// Mitsubishi GX Works2 project: PLC_GROUP_10   PLC: FX3G

// global labels: Global1
VAR_GLOBAL CONSTANT
  spieces_ratio : REAL := 0.1;
END_VAR
VAR_GLOBAL
  spieces_wanted AT D1118 : REAL;
  oil_wanted AT D1114 : REAL;
  water_wanted AT D1116 : REAL;
  yeast_wanted AT D1112 : REAL;
  Enough_yeast AT M11 : BOOL;
  Enough_oil AT M12 : BOOL;
  Enough_spieces AT M14 : BOOL;
  turn_of_flickering AT TC1 : BOOL;
END_VAR
VAR_GLOBAL CONSTANT
  ThreeSec : INT := 30;
END_VAR
VAR_GLOBAL
  blink AT M5 : BOOL;
  TC2 AT TC2 : BOOL;
  TC_2 AT TC2 : BOOL;
END_VAR
VAR_GLOBAL CONSTANT
  half_Sec : INT := 5;
END_VAR
VAR_GLOBAL
  TS_2 AT TS2 : BOOL;
  TC_3 AT TC3 : BOOL;
  TS_3 AT TS3 : BOOL;
  TS_1 AT TS1 : BOOL;
  StatrWork AT X002 : BOOL;
  StartWork AT X002 : BOOL;
  TS_5 AT TS5 : BOOL;
END_VAR
VAR_GLOBAL CONSTANT
  Lamp_on : REAL := 30.0;
END_VAR
VAR_GLOBAL
  TC_5 AT TC5 : BOOL;
  Lamp_Before_work AT Y005 : BOOL;
END_VAR
VAR_GLOBAL CONSTANT
  const100 : REAL := 100.0;
END_VAR
VAR_GLOBAL
  Kneading_flour AT D1300 : REAL;
END_VAR
VAR_GLOBAL CONSTANT
  const20 : REAL := 20.0;
END_VAR
VAR_GLOBAL
  Kneading_yeast AT D1302 : REAL;
END_VAR
VAR_GLOBAL CONSTANT
  const50 : REAL := 50.0;
END_VAR
VAR_GLOBAL
  Kneading_water AT D1306 : REAL;
END_VAR
VAR_GLOBAL CONSTANT
  const30 : REAL := 30.0;
END_VAR
VAR_GLOBAL
  Kneading_oil AT D1304 : REAL;
  Kneading_spieces AT D1308 : REAL;
END_VAR
VAR_GLOBAL CONSTANT
  const10 : REAL := 10.0;
END_VAR
VAR_GLOBAL
  TC_4 AT TC4 : BOOL;
  TS_4 AT TS4 : BOOL;
  Start_kneading AT X001 : BOOL;
  kneading_light AT Y001 : BOOL;
  mix_flour AT D1300 : REAL;
  mix_yeast AT D1302 : REAL;
  mix_water AT D1306 : REAL;
  mix_oil AT D1304 : REAL;
  mix_spieces AT D1308 : REAL;
  rising_flour AT D1400 : REAL;
  rising_yeast AT D1402 : REAL;
  rising_water AT D1406 : REAL;
  rising_oil AT D1404 : REAL;
  rising_spieces AT D1408 : REAL;
  Start_baking AT M9 : BOOL;
  Start_rising AT M100 : BOOL;
  baking_flour AT D1500 : REAL;
  baking_yeast AT D1502 : REAL;
  baking_water AT D1506 : REAL;
  baking_oil AT D1504 : REAL;
  baking_spieces AT D1508 : REAL;
  Start_Mix AT X001 : BOOL;
  Mix_light AT Y001 : BOOL;
  Start_Rising_Dough AT X011 : BOOL;
  Count_Clicks AT CC1 : BOOL;
END_VAR
VAR_GLOBAL CONSTANT
  clicks_2 : INT := 2;
END_VAR
VAR_GLOBAL
  CS_1 AT CS1 : BOOL;
  turn_of_blinking AT TC8 : BOOL;
  TC_8 AT TC8 : BOOL;
  blinking AT M7 : BOOL;
  TC_6 AT TC6 : BOOL;
  TS_6 AT TS6 : BOOL;
  Rising_Light_1 AT Y002 : BOOL;
  TC_7 AT TC7 : BOOL;
  TS_7 AT TS7 : BOOL;
  Rising_Light_2 AT Y003 : BOOL;
  TS_8 AT TS8 : BOOL;
  finish_Raising AT M8 : BOOL;
  finish_Rising AT M8 : BOOL;
  TS_9 AT TS9 : BOOL;
  baking AT Y004 : BOOL;
  EnoughStock AT M2 : BOOL;
  Transfer_ingridients AT M13 : BOOL;
  flour_trasfered AT M15 : BOOL;
  yeast_trasfered AT M16 : BOOL;
  water_trasfered AT M17 : BOOL;
  oil_trasfered AT M18 : BOOL;
  spieces_trasfered AT M19 : BOOL;
  Start_clock AT M20 : BOOL;
  TransferFlour AT M21 : BOOL;
  TransferYeast AT M22 : BOOL;
  TrasnferWater AT M22 : BOOL;
  TransferOil AT M24 : BOOL;
  TransferWater AT M23 : BOOL;
  TransferSpeices AT M25 : BOOL;
  TransferIngridients AT M80 : BOOL;
  StartClock AT M26 : BOOL;
  baking_timer AT TC9 : BOOL;
  TrayonShelf_flour AT D1600 : REAL;
  TrayonShelf_yeast AT D1602 : REAL;
  TrayonShelf_water AT D1606 : REAL;
  TrayonShelf_oil AT D1604 : REAL;
  TrayonShelf_spieces AT D1608 : REAL;
  Transfer_Flour AT M26 : BOOL;
  Transfer_Yeast AT M27 : BOOL;
  Transfer_Water AT M28 : BOOL;
  Transfer_Oil AT M29 : BOOL;
  Transfer_Speices AT M30 : BOOL;
  quality_check AT X003 : BOOL;
  Check_amounts AT CC16 : BOOL;
END_VAR
VAR_GLOBAL CONSTANT
  two_checks : INT := 3;
END_VAR
VAR_GLOBAL
  CS_2 AT CS2 : BOOL;
  Analog_Input_2 AT D8281 : REAL;
END_VAR
VAR_GLOBAL CONSTANT
  LB : INT := 400;
END_VAR
VAR_GLOBAL
  GE_than_1 AT M27 : BOOL;
  LE_than_5 AT M28 : BOOL;
  quality_timer AT TC11 : BOOL;
END_VAR
VAR_GLOBAL CONSTANT
  five_sec : INT := 50;
  UB : INT := 2000;
END_VAR
VAR_GLOBAL
  TS_11 AT TS11 : BOOL;
  quality_light AT Y006 : BOOL;
  ThrowToGarbage AT M30 : BOOL;
END_VAR
VAR_GLOBAL CONSTANT
  const0 : REAL;
  oil_ratio : REAL := 0.3;
  water_ratio : REAL := 0.5;
  yeast_ratio : REAL := 0.2;
  constant_100 : REAL := 100.0;
END_VAR
VAR_GLOBAL
  OutOfStock AT M2 : BOOL;
  EmergencyButton AT X007 : BOOL;
  EndWorkDay AT M10 : BOOL;
  WorkDayLight AT Y010 : BOOL;
  StartDay AT X010 : BOOL;
  spices_stock AT D1208 : REAL;
  spieces_input AT D1108 : REAL;
  spieces_stock AT D1208 : REAL;
  sesame_stock AT D1212 : REAL;
  sesame_input AT D1114 : REAL;
  salt_stock AT D1210 : REAL;
  salt_input AT D1112 : REAL;
  suger_stock AT D1208 : REAL;
  suger_input AT D1110 : REAL;
  water_stock AT D1206 : REAL;
  water_input AT D1106 : REAL;
  oil_stock AT D1204 : REAL;
  oil_input AT D1104 : REAL;
  yeast_stock AT D1202 : REAL;
  yeast_input AT D1102 : REAL;
  flour_input AT D1100 : REAL;
  flour_stock AT D1200 : REAL;
  Switch_start_Day AT X010 : BOOL;
  Lamp_start_work AT Y005 : BOOL;
  Switch1 AT X002 : BOOL;
  Enough_water AT M13 : BOOL;
END_VAR
VAR_GLOBAL CONSTANT
  four_sec : INT := 40;
END_VAR
VAR_GLOBAL
  Steady_light AT M50 : BOOL;
  blinking_light AT M51 : BOOL;
  Mix_active AT M60 : BOOL;
  Counter_light AT M61 : BOOL;
  off_blinkingLight AT M52 : BOOL;
  Check1 AT M80 : BOOL;
  Check2 AT M81 : BOOL;
  Check3 AT M82 : BOOL;
  Check4 AT M83 : BOOL;
  Check5 AT M84 : BOOL;
  yalla AT M100 : BOOL;
  SHAY AT M222 : BOOL;
  closed AT M223 : BOOL;
  RESET_DAY AT M224 : BOOL;
  AnalogInput2 AT D8281 : INT;
END_VAR
VAR_GLOBAL CONSTANT
  LBLB : REAL := 2000.0;
END_VAR
VAR_GLOBAL
  ResetCounter AT M230 : BOOL;
  REalinput AT D8281 : REAL;
  CC_2 AT CC2 : BOOL;
  LB_flour AT M102 : BOOL;
END_VAR
VAR_GLOBAL CONSTANT
  two_checks_forGarbage : INT := 2;
END_VAR
VAR_GLOBAL
  CC_3 AT CC3 : BOOL;
  M_Flour AT M338 : BOOL;
  M_Yeast AT M339 : BOOL;
  M_Water AT M340 : BOOL;
  M_Oil AT M341 : BOOL;
  M_Spieces AT M342 : BOOL;
  M_Flour2 AT M330 : BOOL;
  M_Yeast2 AT M331 : BOOL;
  M_Wate2r AT M332 : BOOL;
  M_Oil2 AT M333 : BOOL;
  M_Spieces2 AT M334 : BOOL;
  M_Wate2 AT M332 : BOOL;
  M_Water2 AT M332 : BOOL;
  finish_it AT M335 : BOOL;
  flour_container AT D1250 : REAL;
  yeast_container AT D1252 : REAL;
  water_container AT D1256 : REAL;
  oil_container AT D1254 : REAL;
  spieces_container AT D1258 : REAL;
  Lamp_Y5Off AT M288 : BOOL;
  UB_twoChecks AT CC2 : BOOL;
  twoChecksForGarbage AT CC3 : BOOL;
  quality_const AT M20 : BOOL;
END_VAR

// task Task_01 (event TRUE, interval 0, priority 31): POU_01

PROGRAM POU_01
(* structured ladder/FBD written out as ST: instructions are called as NAME(EN, inputs, outputs); _pN, _eN, _tN stand for wires *)
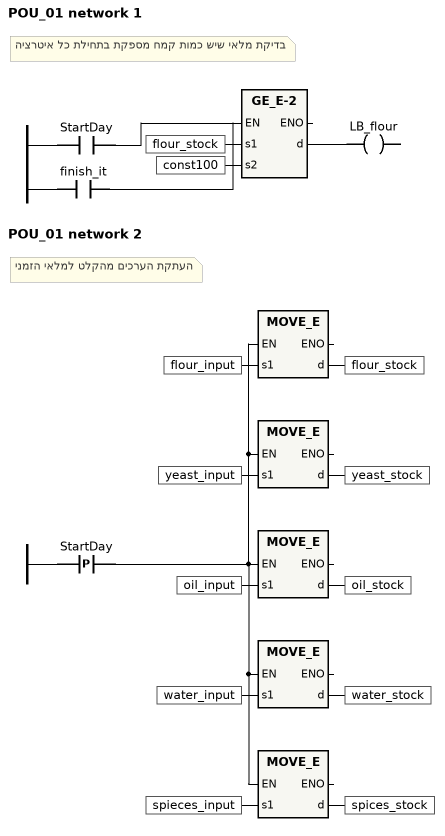
(* network 1 *)
(* בדיקת מלאי שיש כמות קמח מספקת בתחילת כל איטרציה *)
GE_E(StartDay OR finish_it, flour_stock, const100, _t1);
LB_flour := _t1;
(* network 2 *)
(* העתקת הערכים מהקלט למלאי הזמני *)
_p1 := LDP(TRUE, StartDay);
MOVE_E(_p1, flour_input, flour_stock);
MOVE_E(_p1, yeast_input, yeast_stock);
MOVE_E(_p1, oil_input, oil_stock);
MOVE_E(_p1, water_input, water_stock);
MOVE_E(_p1, spieces_input, spices_stock);
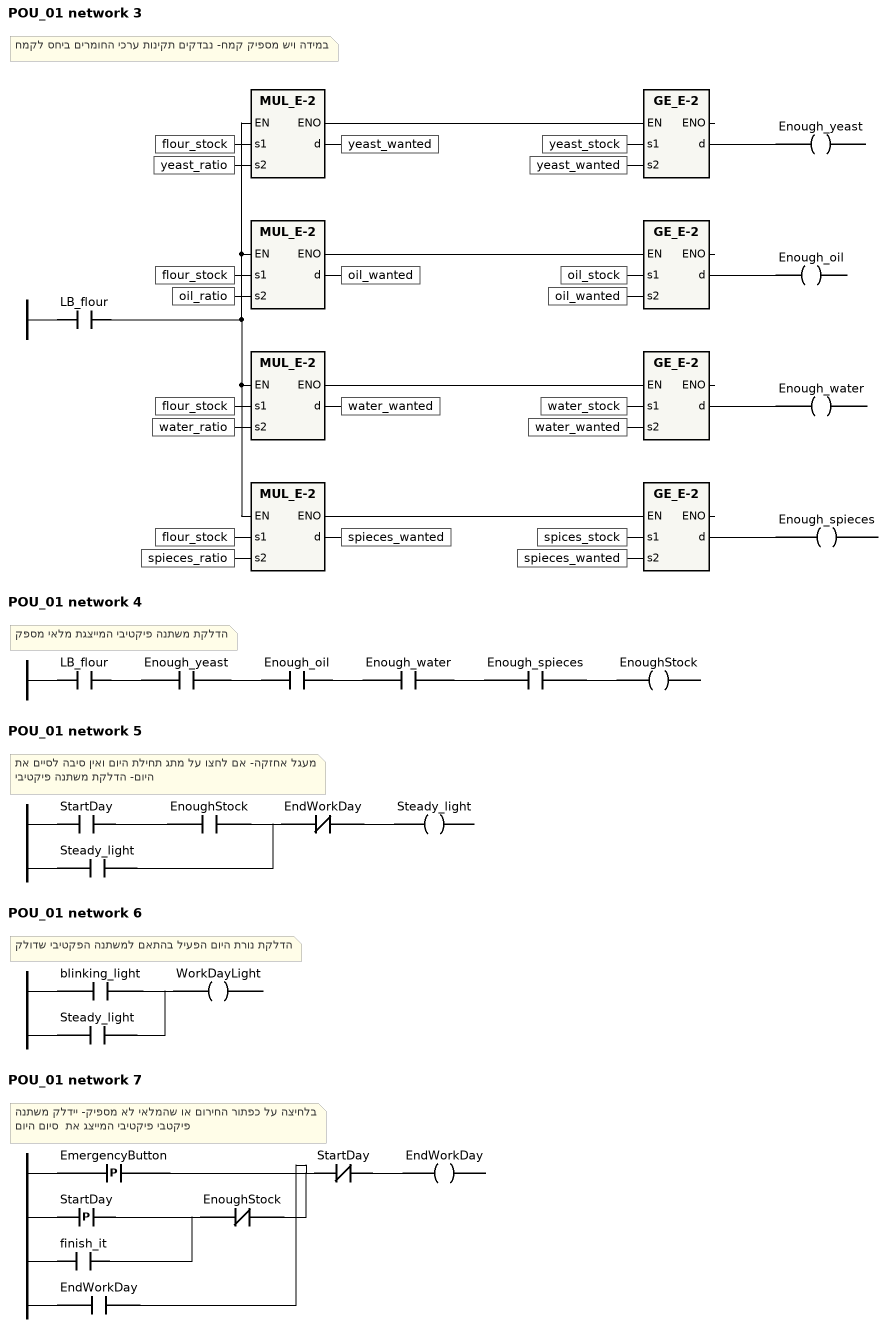
(* network 3 *)
(* במידה ויש מספיק קמח- נבדקים תקינות ערכי החומרים ביחס לקמח *)
_e1 := MUL_E(LB_flour, flour_stock, yeast_ratio, yeast_wanted);
GE_E(_e1, yeast_stock, yeast_wanted, _t2);
Enough_yeast := _t2;
_e3 := MUL_E(LB_flour, flour_stock, oil_ratio, oil_wanted);
GE_E(_e3, oil_stock, oil_wanted, _t4);
Enough_oil := _t4;
_e5 := MUL_E(LB_flour, flour_stock, water_ratio, water_wanted);
GE_E(_e5, water_stock, water_wanted, _t6);
Enough_water := _t6;
_e7 := MUL_E(LB_flour, flour_stock, spieces_ratio, spieces_wanted);
GE_E(_e7, spices_stock, spieces_wanted, _t8);
Enough_spieces := _t8;
(* network 4 *)
(* הדלקת משתנה פיקטיבי המייצגת מלאי מספק *)
EnoughStock := LB_flour AND Enough_yeast AND Enough_oil AND Enough_water AND Enough_spieces;
(* network 5 *)
(* מעגל אחזקה- אם לחצו על מתג תחילת היום ואין סיבה לסיים את היום- הדלקת משתנה פיקטיבי *)
Steady_light := ((StartDay AND EnoughStock) OR Steady_light) AND NOT EndWorkDay;
(* network 6 *)
(* הדלקת נורת היום הפעיל בהתאם למשתנה הפקטיבי שדולק *)
WorkDayLight := blinking_light OR Steady_light;
(* network 7 *)
(* בלחיצה על כפתור החירום או שהמלאי לא מספיק- יידלק משתנה פיקטבי פיקטיבי המייצג את  סיום היום *)
EndWorkDay := (LDP(TRUE, EmergencyButton) OR ((LDP(TRUE, StartDay) OR finish_it) AND NOT EnoughStock) OR EndWorkDay) AND NOT StartDay;
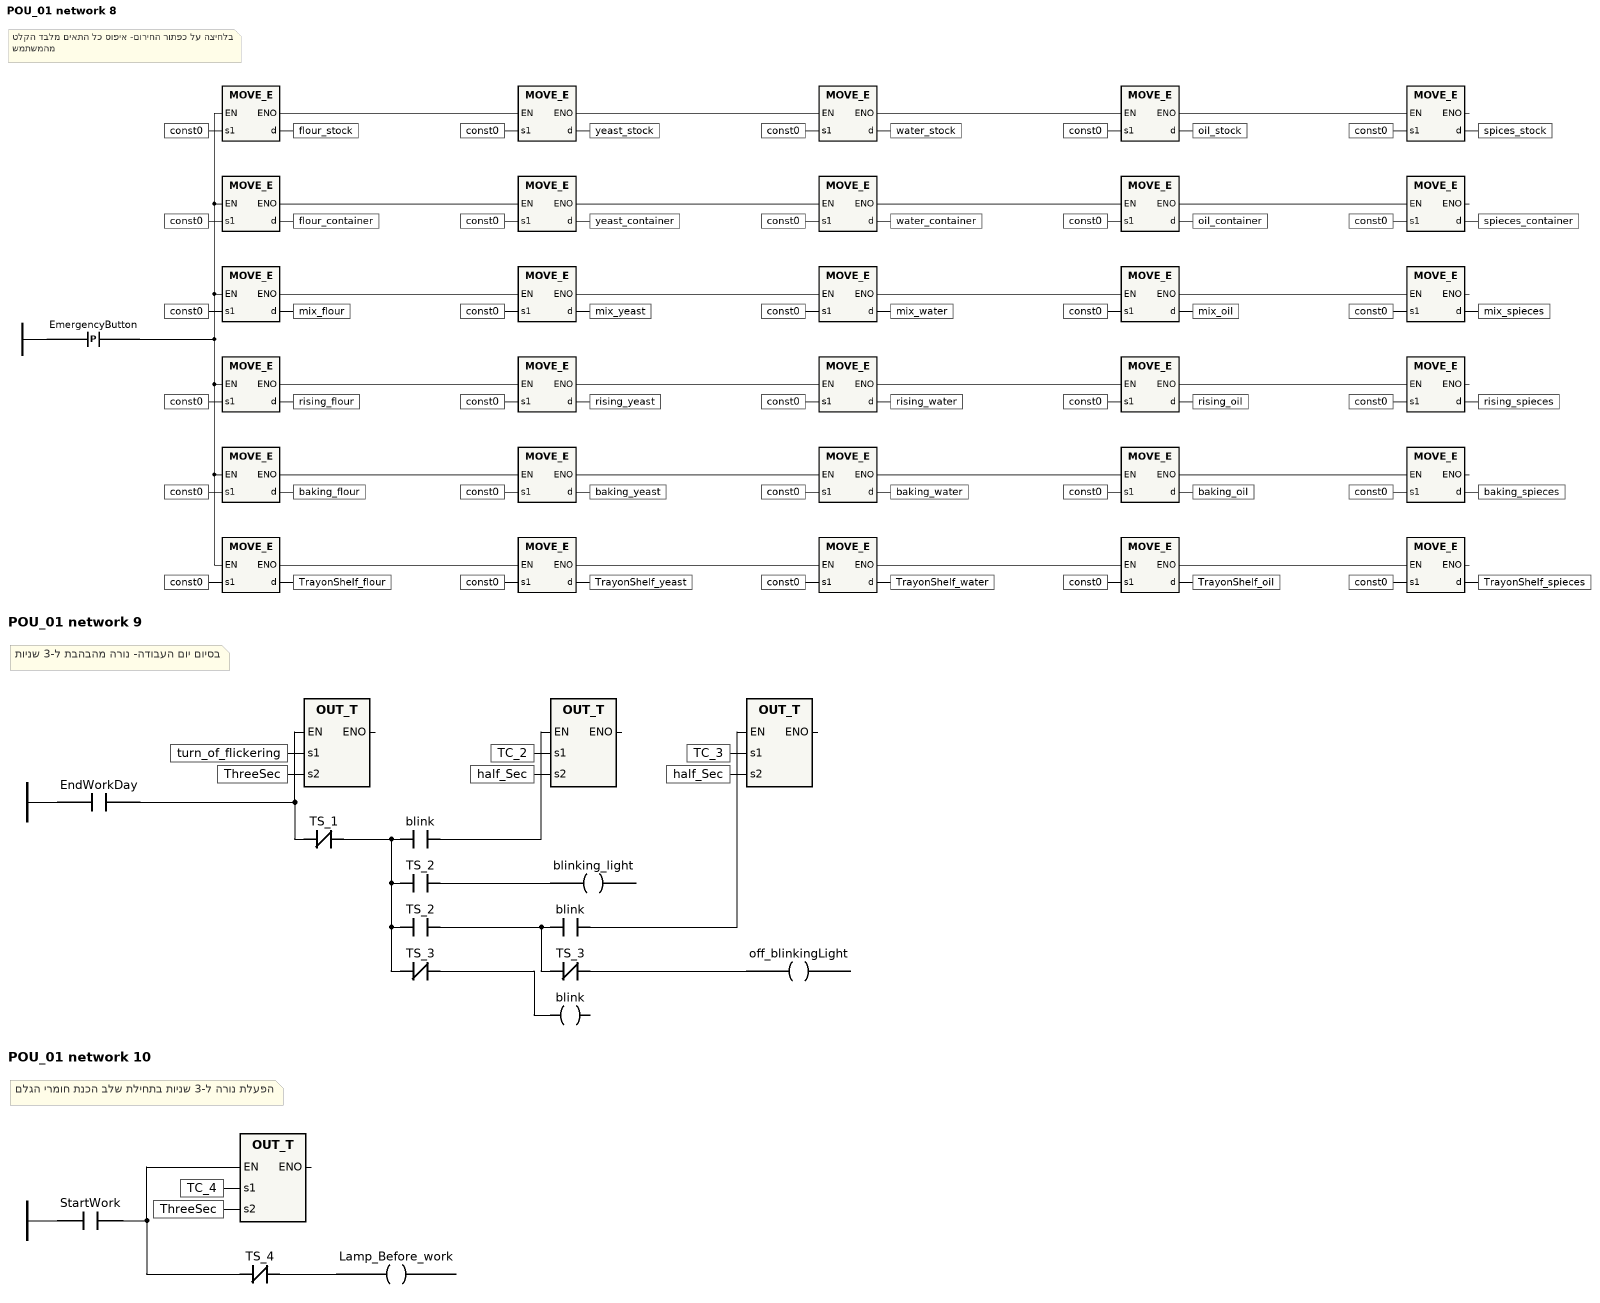
(* network 8 *)
(* בלחיצה על כפתור החירום- איפוס כל התאים מלבד הקלט מהמשתמש *)
_p1 := LDP(TRUE, EmergencyButton);
_e2 := MOVE_E(_p1, const0, flour_stock);
_e3 := MOVE_E(_e2, const0, yeast_stock);
_e4 := MOVE_E(_e3, const0, water_stock);
_e5 := MOVE_E(_e4, const0, oil_stock);
MOVE_E(_e5, const0, spices_stock);
_e6 := MOVE_E(_p1, const0, flour_container);
_e7 := MOVE_E(_e6, const0, yeast_container);
_e8 := MOVE_E(_e7, const0, water_container);
_e9 := MOVE_E(_e8, const0, oil_container);
MOVE_E(_e9, const0, spieces_container);
_e10 := MOVE_E(_p1, const0, mix_flour);
_e11 := MOVE_E(_e10, const0, mix_yeast);
_e12 := MOVE_E(_e11, const0, mix_water);
_e13 := MOVE_E(_e12, const0, mix_oil);
MOVE_E(_e13, const0, mix_spieces);
_e14 := MOVE_E(_p1, const0, rising_flour);
_e15 := MOVE_E(_e14, const0, rising_yeast);
_e16 := MOVE_E(_e15, const0, rising_water);
_e17 := MOVE_E(_e16, const0, rising_oil);
MOVE_E(_e17, const0, rising_spieces);
_e18 := MOVE_E(_p1, const0, baking_flour);
_e19 := MOVE_E(_e18, const0, baking_yeast);
_e20 := MOVE_E(_e19, const0, baking_water);
_e21 := MOVE_E(_e20, const0, baking_oil);
MOVE_E(_e21, const0, baking_spieces);
_e22 := MOVE_E(_p1, const0, TrayonShelf_flour);
_e23 := MOVE_E(_e22, const0, TrayonShelf_yeast);
_e24 := MOVE_E(_e23, const0, TrayonShelf_water);
_e25 := MOVE_E(_e24, const0, TrayonShelf_oil);
MOVE_E(_e25, const0, TrayonShelf_spieces);
(* network 9 *)
(* בסיום יום העבודה- נורה מהבהבת ל-3 שניות *)
OUT_T(EndWorkDay, turn_of_flickering, ThreeSec);
_p1 := EndWorkDay AND NOT TS_1;
OUT_T(_p1 AND blink, TC_2, half_Sec);
blinking_light := _p1 AND TS_2;
_p2 := _p1 AND TS_2;
OUT_T(_p2 AND blink, TC_3, half_Sec);
off_blinkingLight := _p2 AND NOT TS_3;
blink := _p1 AND NOT TS_3;
(* network 10 *)
(* הפעלת נורה ל-3 שניות בתחילת שלב הכנת חומרי הגלם *)
OUT_T(StartWork, TC_4, ThreeSec);
Lamp_Before_work := StartWork AND NOT TS_4;
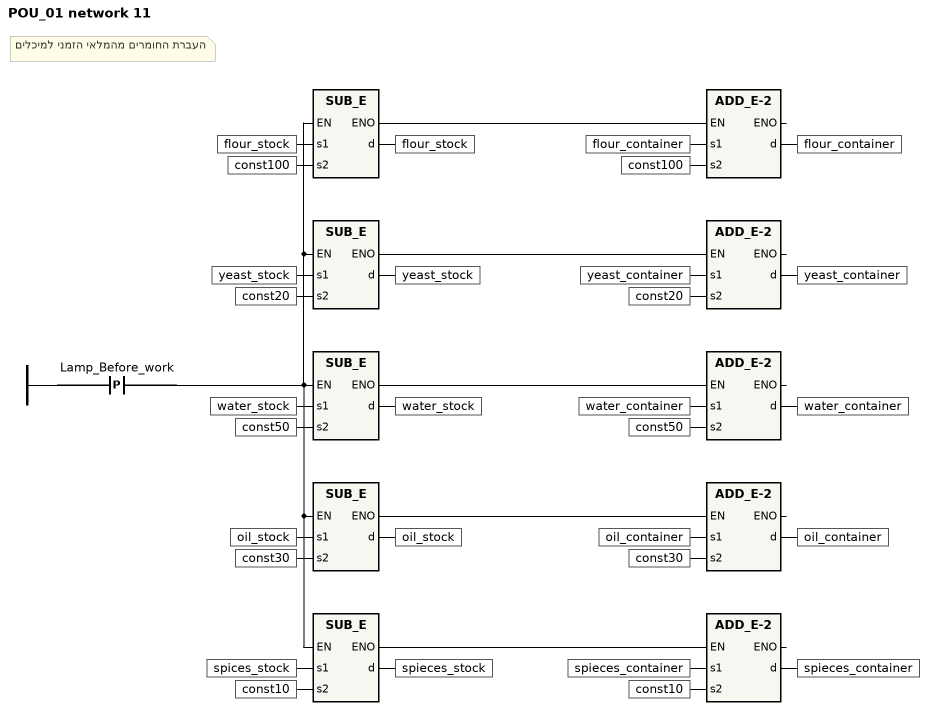
(* network 11 *)
(* העברת החומרים מהמלאי הזמני למיכלים *)
_p1 := LDP(TRUE, Lamp_Before_work);
_e2 := SUB_E(_p1, flour_stock, const100, flour_stock);
ADD_E(_e2, flour_container, const100, flour_container);
_e3 := SUB_E(_p1, yeast_stock, const20, yeast_stock);
ADD_E(_e3, yeast_container, const20, yeast_container);
_e4 := SUB_E(_p1, water_stock, const50, water_stock);
ADD_E(_e4, water_container, const50, water_container);
_e5 := SUB_E(_p1, oil_stock, const30, oil_stock);
ADD_E(_e5, oil_container, const30, oil_container);
_e6 := SUB_E(_p1, spices_stock, const10, spieces_stock);
ADD_E(_e6, spieces_container, const10, spieces_container);
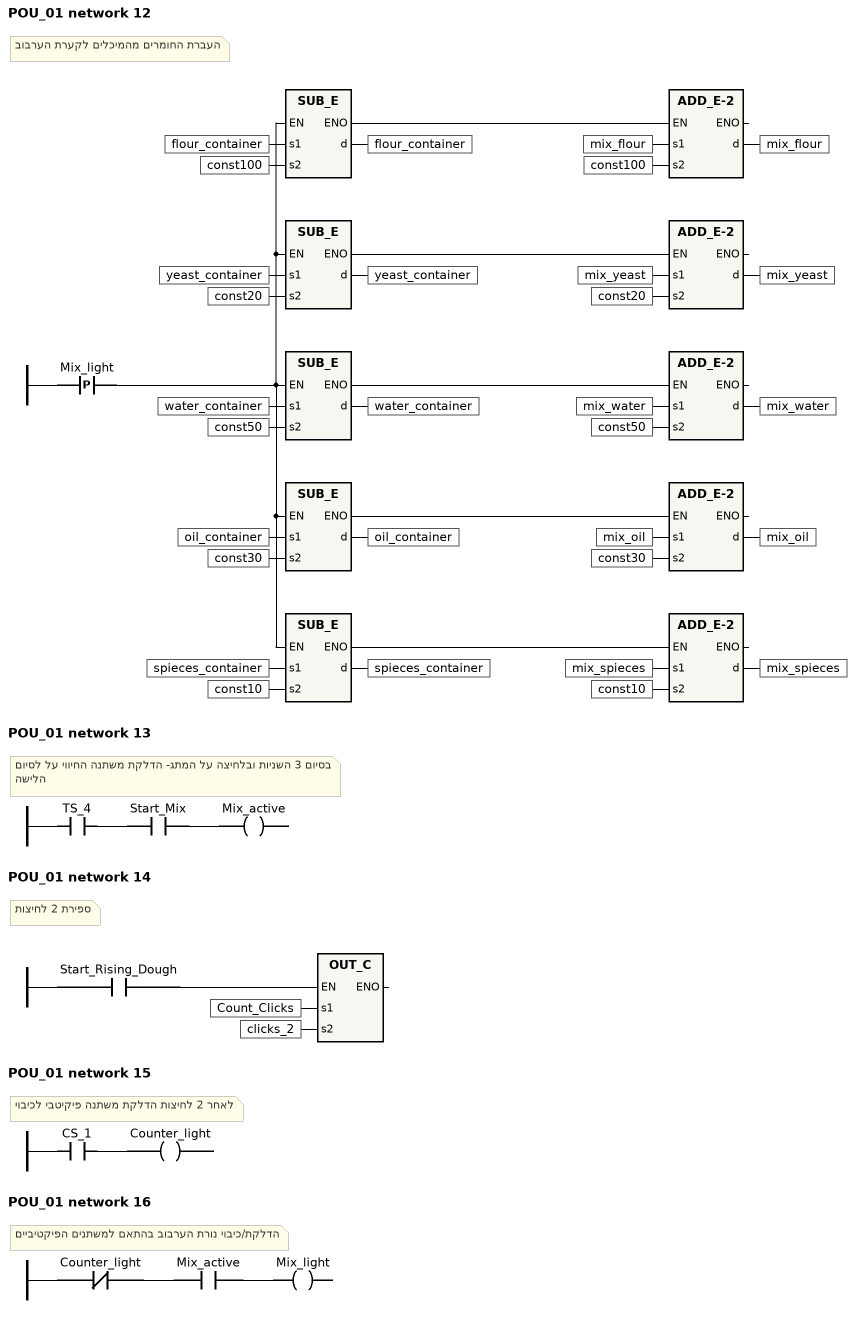
(* network 12 *)
(* העברת החומרים מהמיכלים לקערת הערבוב *)
_p1 := LDP(TRUE, Mix_light);
_e2 := SUB_E(_p1, flour_container, const100, flour_container);
ADD_E(_e2, mix_flour, const100, mix_flour);
_e3 := SUB_E(_p1, yeast_container, const20, yeast_container);
ADD_E(_e3, mix_yeast, const20, mix_yeast);
_e4 := SUB_E(_p1, water_container, const50, water_container);
ADD_E(_e4, mix_water, const50, mix_water);
_e5 := SUB_E(_p1, oil_container, const30, oil_container);
ADD_E(_e5, mix_oil, const30, mix_oil);
_e6 := SUB_E(_p1, spieces_container, const10, spieces_container);
ADD_E(_e6, mix_spieces, const10, mix_spieces);
(* network 13 *)
(* בסיום 3 השניות ובלחיצה על המתג- הדלקת משתנה החיווי על לסיום הלישה *)
Mix_active := TS_4 AND Start_Mix;
(* network 14 *)
(* ספירת 2 לחיצות *)
OUT_C(Start_Rising_Dough, Count_Clicks, clicks_2);
(* network 15 *)
(* לאחר 2 לחיצות הדלקת משתנה פיקיטבי לכיבוי *)
Counter_light := CS_1;
(* network 16 *)
(* הדלקת/כיבוי נורת הערבוב בהתאם למשתנים הפיקטיביים *)
Mix_light := NOT Counter_light AND Mix_active;
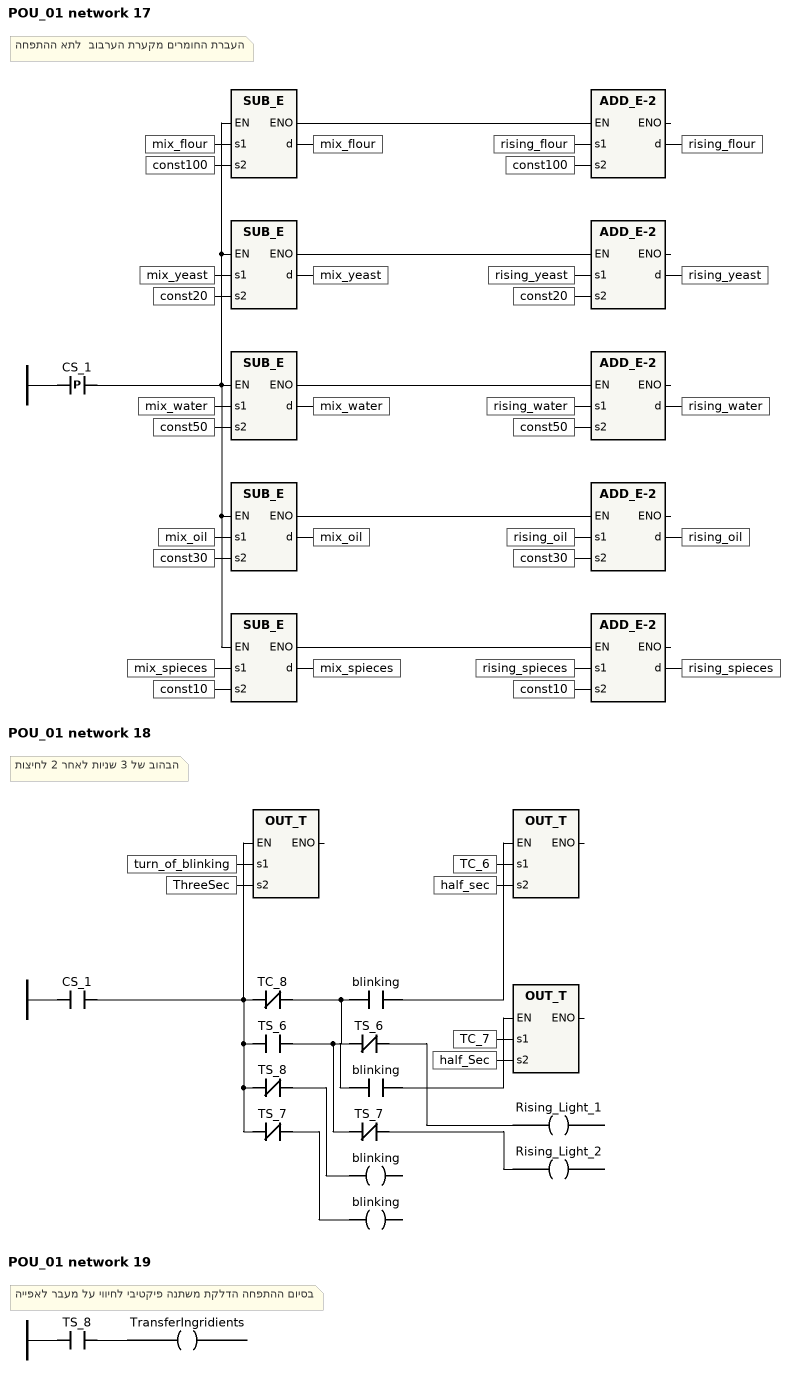
(* network 17 *)
(* העברת החומרים מקערת הערבוב  לתא ההתפחה *)
_p1 := LDP(TRUE, CS_1);
_e2 := SUB_E(_p1, mix_flour, const100, mix_flour);
ADD_E(_e2, rising_flour, const100, rising_flour);
_e3 := SUB_E(_p1, mix_yeast, const20, mix_yeast);
ADD_E(_e3, rising_yeast, const20, rising_yeast);
_e4 := SUB_E(_p1, mix_water, const50, mix_water);
ADD_E(_e4, rising_water, const50, rising_water);
_e5 := SUB_E(_p1, mix_oil, const30, mix_oil);
ADD_E(_e5, rising_oil, const30, rising_oil);
_e6 := SUB_E(_p1, mix_spieces, const10, mix_spieces);
ADD_E(_e6, rising_spieces, const10, rising_spieces);
(* network 18 *)
(* הבהוב של 3 שניות לאחר 2 לחיצות *)
OUT_T(CS_1, turn_of_blinking, ThreeSec);
_p1 := CS_1 AND NOT TC_8;
OUT_T(_p1 AND blinking, TC_6, half_sec);
Rising_Light_1 := _p1 AND NOT TS_6;
_p2 := CS_1 AND TS_6;
OUT_T(_p2 AND blinking, TC_7, half_Sec);
Rising_Light_2 := _p2 AND NOT TS_7;
blinking := CS_1 AND NOT TS_8;
blinking := CS_1 AND NOT TS_7;
(* network 19 *)
(* בסיום ההתפחה הדלקת משתנה פיקטיבי לחיווי על מעבר לאפייה *)
TransferIngridients := TS_8;
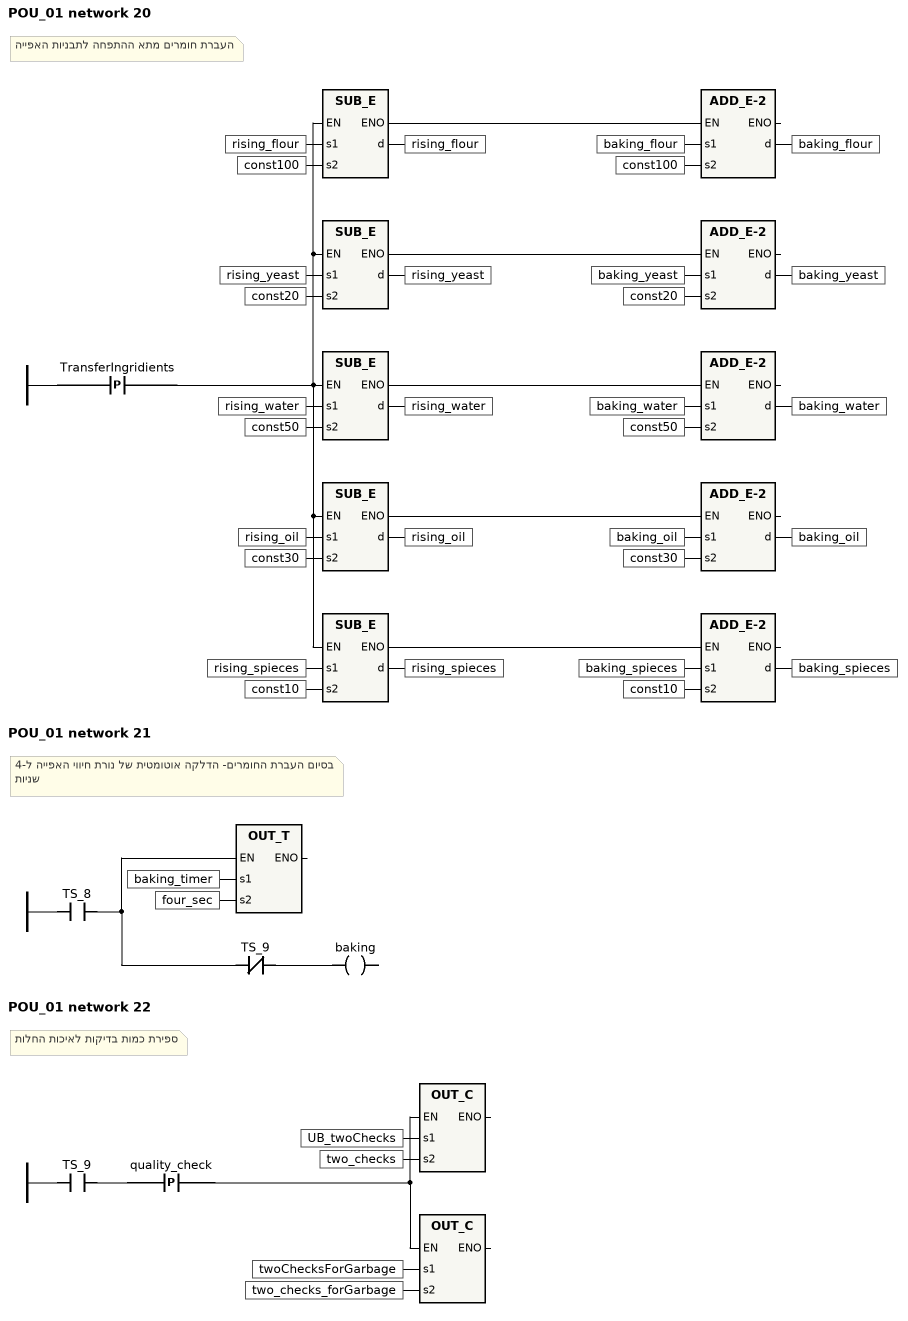
(* network 20 *)
(* העברת חומרים מתא ההתפחה לתבניות האפייה *)
_p1 := LDP(TRUE, TransferIngridients);
_e2 := SUB_E(_p1, rising_flour, const100, rising_flour);
ADD_E(_e2, baking_flour, const100, baking_flour);
_e3 := SUB_E(_p1, rising_yeast, const20, rising_yeast);
ADD_E(_e3, baking_yeast, const20, baking_yeast);
_e4 := SUB_E(_p1, rising_water, const50, rising_water);
ADD_E(_e4, baking_water, const50, baking_water);
_e5 := SUB_E(_p1, rising_oil, const30, rising_oil);
ADD_E(_e5, baking_oil, const30, baking_oil);
_e6 := SUB_E(_p1, rising_spieces, const10, rising_spieces);
ADD_E(_e6, baking_spieces, const10, baking_spieces);
(* network 21 *)
(* בסיום העברת החומרים- הדלקה אוטומטית של נורת חיווי האפייה ל-4 שניות *)
OUT_T(TS_8, baking_timer, four_sec);
baking := TS_8 AND NOT TS_9;
(* network 22 *)
(* ספירת כמות בדיקות לאיכות החלות *)
_p1 := TS_9 AND LDP(TRUE, quality_check);
OUT_C(_p1, UB_twoChecks, two_checks);
OUT_C(_p1, twoChecksForGarbage, two_checks_forGarbage);
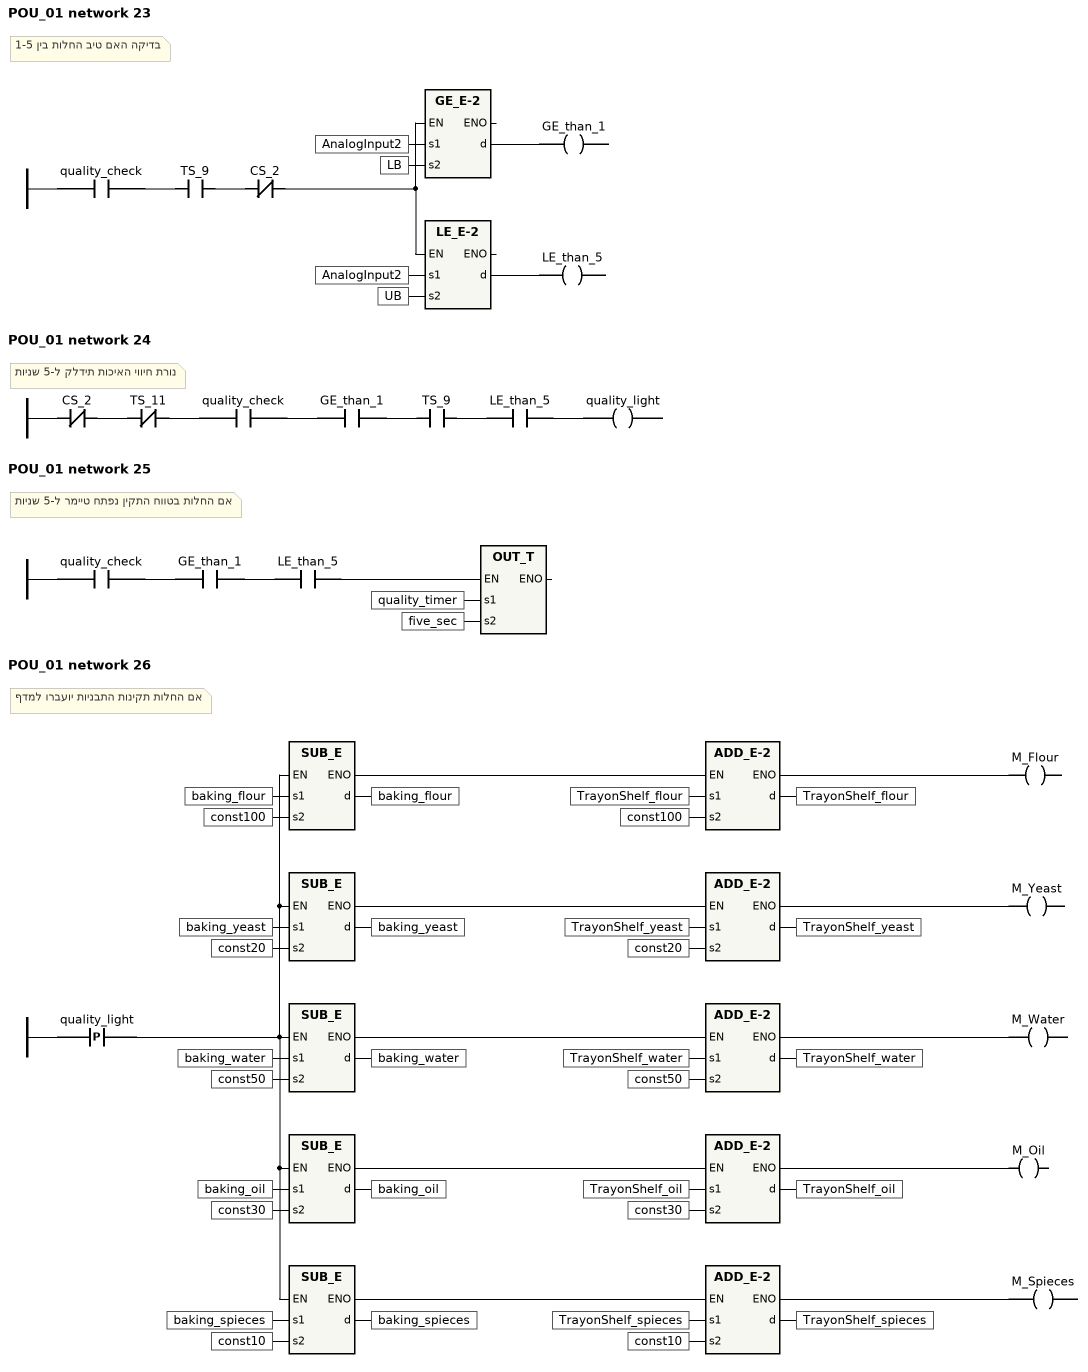
(* network 23 *)
(* בדיקה האם טיב החלות בין 1-5 *)
_p1 := quality_check AND TS_9 AND NOT CS_2;
GE_E(_p1, AnalogInput2, LB, _t2);
GE_than_1 := _t2;
LE_E(_p1, AnalogInput2, UB, _t3);
LE_than_5 := _t3;
(* network 24 *)
(* נורת חיווי האיכות תידלק ל-5 שניות *)
quality_light := NOT CS_2 AND NOT TS_11 AND quality_check AND GE_than_1 AND TS_9 AND LE_than_5;
(* network 25 *)
(* אם החלות בטווח התקין נפתח טיימר ל-5 שניות *)
OUT_T(quality_check AND GE_than_1 AND LE_than_5, quality_timer, five_sec);
(* network 26 *)
(* אם החלות תקינות התבניות יועברו למדף *)
_p1 := LDP(TRUE, quality_light);
_e2 := SUB_E(_p1, baking_flour, const100, baking_flour);
_e3 := ADD_E(_e2, TrayonShelf_flour, const100, TrayonShelf_flour);
M_Flour := _e3;
_e4 := SUB_E(_p1, baking_yeast, const20, baking_yeast);
_e5 := ADD_E(_e4, TrayonShelf_yeast, const20, TrayonShelf_yeast);
M_Yeast := _e5;
_e6 := SUB_E(_p1, baking_water, const50, baking_water);
_e7 := ADD_E(_e6, TrayonShelf_water, const50, TrayonShelf_water);
M_Water := _e7;
_e8 := SUB_E(_p1, baking_oil, const30, baking_oil);
_e9 := ADD_E(_e8, TrayonShelf_oil, const30, TrayonShelf_oil);
M_Oil := _e9;
_e10 := SUB_E(_p1, baking_spieces, const10, baking_spieces);
_e11 := ADD_E(_e10, TrayonShelf_spieces, const10, TrayonShelf_spieces);
M_Spieces := _e11;
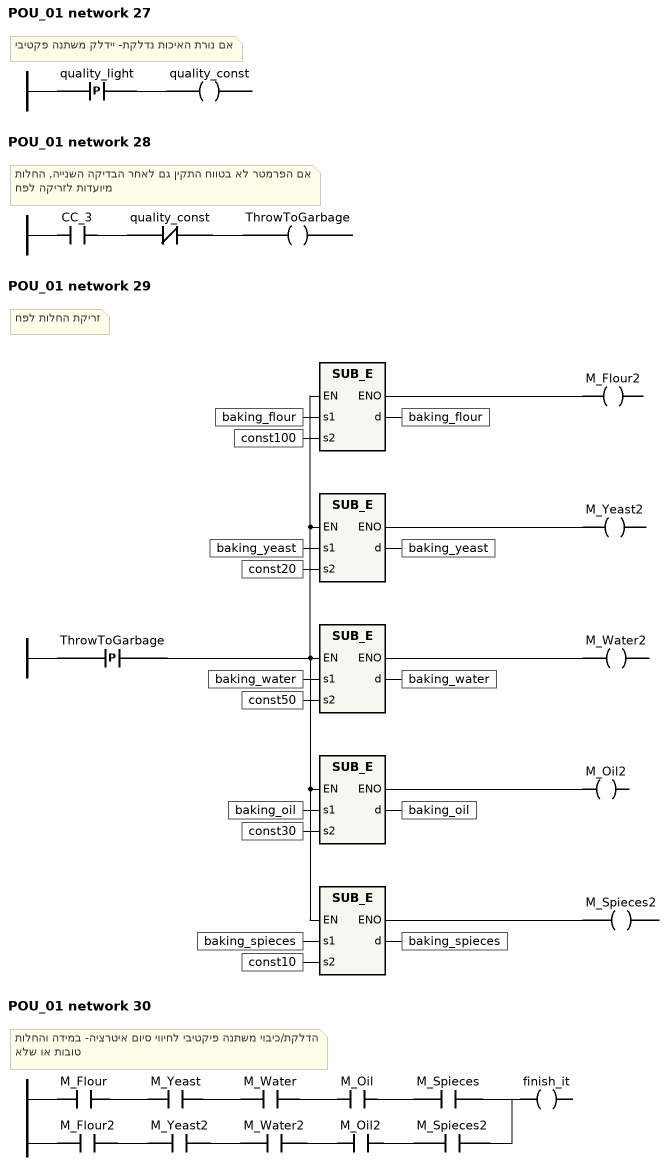
(* network 27 *)
(* אם נורת האיכות נדלקת- יידלק משתנה פקטיבי *)
quality_const := LDP(TRUE, quality_light);
(* network 28 *)
(* אם הפרמטר לא בטווח התקין גם לאחר הבדיקה השנייה, החלות מיועדות לזריקה לפח *)
ThrowToGarbage := CC_3 AND NOT quality_const;
(* network 29 *)
(* זריקת החלות לפח *)
_p1 := LDP(TRUE, ThrowToGarbage);
_e2 := SUB_E(_p1, baking_flour, const100, baking_flour);
M_Flour2 := _e2;
_e3 := SUB_E(_p1, baking_yeast, const20, baking_yeast);
M_Yeast2 := _e3;
_e4 := SUB_E(_p1, baking_water, const50, baking_water);
M_Water2 := _e4;
_e5 := SUB_E(_p1, baking_oil, const30, baking_oil);
M_Oil2 := _e5;
_e6 := SUB_E(_p1, baking_spieces, const10, baking_spieces);
M_Spieces2 := _e6;
(* network 30 *)
(* הדלקת/כיבוי משתנה פיקטיבי לחיווי סיום איטרציה- במידה והחלות טובות או שלא *)
finish_it := (M_Flour AND M_Yeast AND M_Water AND M_Oil AND M_Spieces) OR (M_Flour2 AND M_Yeast2 AND M_Water2 AND M_Oil2 AND M_Spieces2);
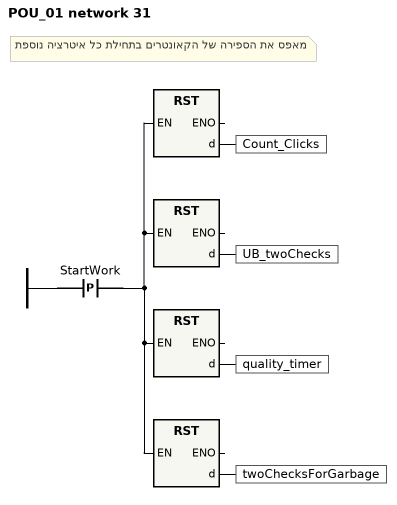
(* network 31 *)
(* מאפס את הספירה של הקאונטרים בתחילת כל איטרציה נוספת *)
_p1 := LDP(TRUE, StartWork);
RST(_p1, Count_Clicks);
RST(_p1, UB_twoChecks);
RST(_p1, quality_timer);
RST(_p1, twoChecksForGarbage);
END_PROGRAM
